// TIA Portal V20 export
DATA_BLOCK "BK32"   // DB259
// stored: MemoryReserve 100
   VAR
      "CATHODE MAIN P&P1 VACUUM ON" : Bool := FALSE;
      "CATHODE MAIN P&P1 VACUUM OFF" : Bool := FALSE;
      "CATHODE MAIN P&P2 VACUUM ON" : Bool := FALSE;
      "CATHODE MAIN P&P2 VACUUM OFF" : Bool := FALSE;
      "CATHODE MAIN NG P&P VACUUM ON" : Bool := FALSE;
      "CATHODE MAIN NG P&P VACUUM OFF" : Bool := FALSE;
      "CATHODE ALIGN TABLE VACUUM ON" : Bool := FALSE;
      "CATHODE ALIGN TABLE VACUUM OFF" : Bool := FALSE;
   END_VAR
BEGIN
END_DATA_BLOCK
